FUNCTION_BLOCK FB_LogName IMPLEMENTS I_VisitModules
VAR
END_VAR

METHOD VisitModules
VAR_INPUT
	Module	: I_Module;
END_VAR
ADSLOGSTR(ADSLOG_MSGTYPE_HINT OR ADSLOG_MSGTYPE_LOG, 'The Module Name is: %s', Module.Name);
END_METHOD

END_FUNCTION_BLOCK

(* stored: Version 1.1.0.1, ProductVersion 3.1.4024.12
   POU FB_LogName: Id {1b47ed67-7d23-44be-b576-8de094e1ade3}, SpecialFunc None
   Method VisitModules: Id {82750c65-5245-4f4f-ae88-a050f7f34916} *)
